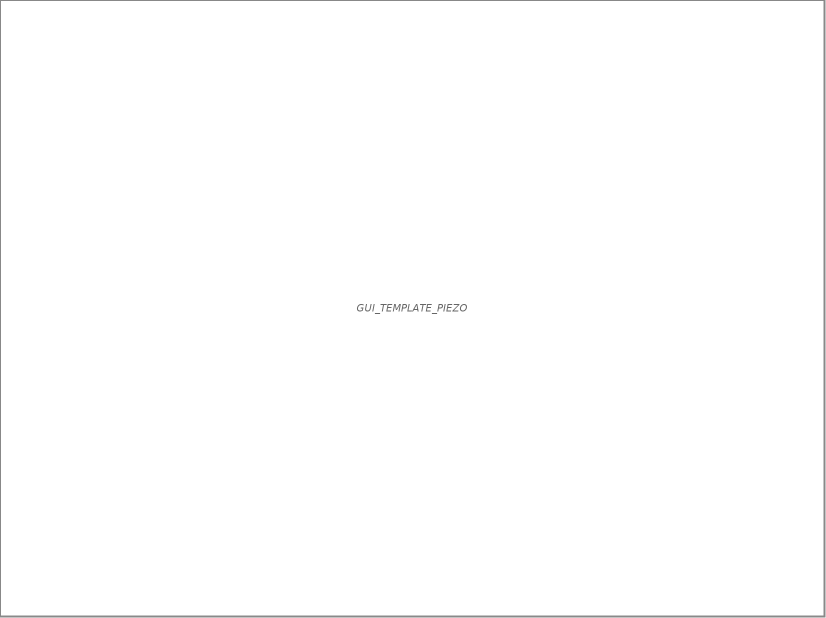
VISUALIZATION GUI_Piezo001  // 826x618
    Frame (0,0 824x616)
        shows GUI_TEMPLATE_PIEZO(m_Instance := MAIN.Piezo001)
END_VISUALIZATION

(* stored: Version 1.1.0.1, ProductVersion 3.1.4024.3
   Visu GUI_Piezo001: Id {3828e674-88ad-4249-8006-fa2151f4bd03} *)
